// TIA Portal V19 export
FUNCTION "AFC_Counter" : Void   // FC1, FBD
TITLE = AFC_COUNTER
{ S7_Optimized_Access := 'TRUE' }
AUTHOR : CH
FAMILY : Aktina
NAME : Global
// AFC_COUNTER
// stored: AutoNumber false, IsIECCheckEnabled true, SetENOAutomatically false
   VAR_INPUT
      Trigger : Bool;
      Pulse : Bool;
      Reset : Bool;
   END_VAR
   VAR_IN_OUT
      Data : Variant;
   END_VAR
   VAR_TEMP
      i : "UDT_COUNTER";
      logical1 : Bool;
   END_VAR
BEGIN

REGION Network 1: GEN: Set Logical 1
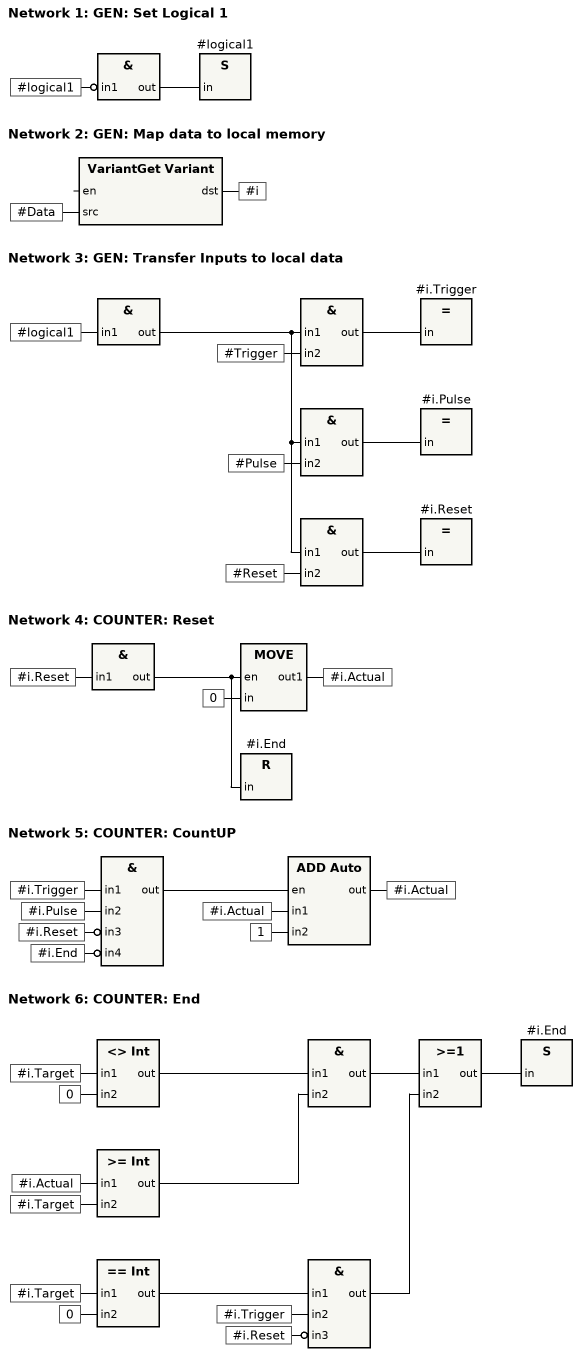
   IF NOT #logical1 THEN #logical1 := TRUE; END_IF;
END_REGION

REGION Network 2: GEN: Map data to local memory
   // no SCL statement known for VariantGet: written as a call
   VariantGet(src := #Data, dst => #i);
END_REGION

REGION Network 3: GEN: Transfer Inputs to local data
   #i.Trigger := #logical1 AND #Trigger;
   #i.Pulse := #logical1 AND #Pulse;
   #i.Reset := #logical1 AND #Reset;
END_REGION

REGION Network 4: COUNTER: Reset
   IF #i.Reset THEN
       #i.Actual := 0;
       #i.End := FALSE;
   END_IF;
END_REGION

REGION Network 5: COUNTER: CountUP
   IF #i.Trigger AND #i.Pulse AND NOT #i.Reset AND NOT #i.End THEN #i.Actual := #i.Actual + 1; END_IF;
END_REGION

REGION Network 6: COUNTER: End
   IF ((#i.Target <> 0) AND (#i.Actual >= #i.Target)) OR ((#i.Target = 0) AND #i.Trigger AND NOT #i.Reset) THEN
       #i.End := TRUE;
   END_IF;
END_REGION

REGION Network 7: COUNTER: Calculate Remaining
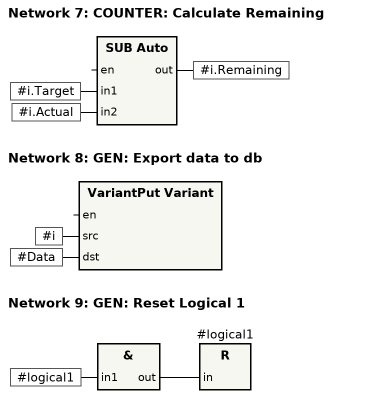
   #i.Remaining := #i.Target - #i.Actual;
END_REGION

REGION Network 8: GEN: Export data to db
   // no SCL statement known for VariantPut: written as a call
   VariantPut(src := #i, dst := #Data);
END_REGION

REGION Network 9: GEN: Reset Logical 1
   IF #logical1 THEN #logical1 := FALSE; END_IF;
END_REGION
END_FUNCTION
